SUBAPPLICATION Uebung_010a4_AX (* SoftKey_F1 auf DigitalOutput_Q1 (Datapanel) *)
  (* Standard: 61499-2; Description: Copyright (c) 2026 Meisterschulen am Ostbahnhof This program and the accompanying materials are made available under the terms of the Eclipse Public License 2.0 which is available at https://www.eclipse.org/legal/epl-2.0/ SPDX-License-Identifier: EPL-2.0 *)
  (* Version 1.0, 2026-01-14, Moritz Ortmeier, Meisterschulen am Ostbahnhof *)
  PACKAGE Uebungen;
  IMPORT DataPanel::io::MI::DQ::DataPanel_MI_DO::DigitalOutput_1A;
  IMPORT DataPanel::io::MI::const::MI::MI_00;
  IMPORT Uebungen::const::UT::DefaultPool::SoftKey_F1;
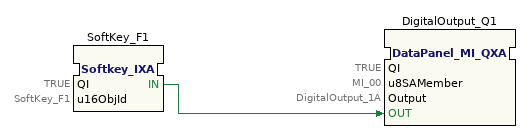
  FBS
    DigitalOutput_Q1 : DataPanel::io::MI::DQ::DataPanel_MI_QXA(QI := TRUE, u8SAMember := MI_00, Output := DigitalOutput_1A);
    SoftKey_F1 : isobus::UT::io::Softkey::Softkey_IXA(QI := TRUE, u16ObjId := SoftKey_F1);
  END_FBS
  ADAPTER_CONNECTIONS
    SoftKey_F1.IN TO DigitalOutput_Q1.OUT;
  END_CONNECTIONS
END_SUBAPPLICATION
